{attribute 'qualified_only'}
VAR_GLOBAL
	Settings: ARRAY[1..100] OF S_Setting;
END_VAR

(* stored: Version 1.1.0.1, ProductVersion 3.1.4024.0
   GVL sp: Id {75bac018-1a5b-4d55-be6f-2c8bf6cba5de} *)
